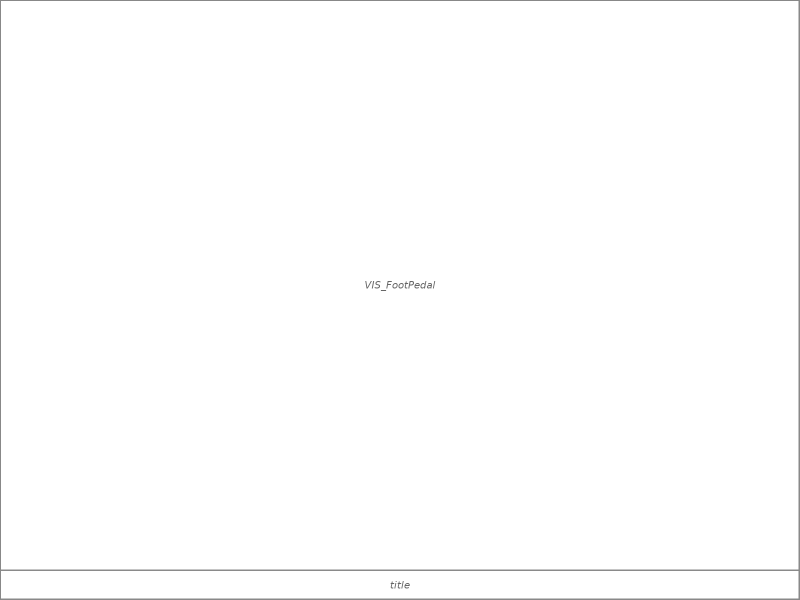
VISUALIZATION F4_System  // 800x600
    TabControl (0,0 800x570)
        shows VIS_FootPedal()
        shows VIS_SaftyGuard()
        shows VIS_SystemEnvironment()
        [0]: TabTitle=FootPedal
        [1]: TabTitle=SaftyGuard
        [2]: TabTitle=Environment
    Frame (0,570 800x30)
        shows title()
END_VISUALIZATION

(* stored: Version 1.1.0.1, ProductVersion 3.1.4024.11
   Visu F4_System: Id {8952a702-d7e4-43a2-a10f-1167f88620eb} *)
